FUNCTION_BLOCK Archive EXTENDS Component
VAR
//	_name : STRING;
	_size : INT;
END_VAR

METHOD AddChild
VAR_INPUT
	Child : I_Component;
END_VAR
END_METHOD

METHOD FB_init : BOOL
VAR_INPUT
	bInitRetains : BOOL; // if TRUE, the retain variables are initialized (warm start / cold start)
	bInCopyCode : BOOL;  // if TRUE, the instance afterwards gets moved into the copy code (online change)
	name : STRING;
	iSize : INT;
END_VAR
THIS^._name := name;
THIS^._size := iSize;
END_METHOD

METHOD GetChildren : ARRAY [1..Param.NumberOfChildren] OF I_Component;
VAR_INPUT
END_VAR
END_METHOD

PROPERTY GetSize : INT
GET
GetSize := _size;
END_GET
END_PROPERTY

END_FUNCTION_BLOCK

(* stored: Version 1.1.0.1, ProductVersion 3.1.4024.12
   POU Archive: Id {5d810e9c-c0b5-44ba-9d2a-66364c59cddb}, SpecialFunc None
   Folder Constructor: Id {1c01b9d4-d31a-4a00-bc33-52a2d495960e}
   Method AddChild: Id {241d4839-b5ce-4c3b-b767-5ff52cc4623c}
   Method FB_init: Id {40a15667-0b65-4fc1-8a61-7083921573ca}
   Method GetChildren: Id {fee8323e-a33a-439d-b512-cf651b3adae1}
   Property GetSize: Id {ff9423c4-8858-49c2-8227-c4fc29b0bf7d}
   Get Get: Id {ade891ab-77fb-466a-af97-f278a6950768} *)
